INTERFACE ITF_Group1 EXTENDS ITF_BaseGroupElement

END_INTERFACE

(* stored: Version 1.1.0.1
   Itf ITF_Group1: Id {2fcbe658-e50b-0a1f-0267-7e71a3ab3742} *)
